FUNCTION_BLOCK E_D_FF_ANY_HYS_TMIN (* Data latch (d) flip flop with a Hysteresis, with a Minimum inter-disposal Time between EO *)
  (* Standard: 61499-1 Annex A; Description: Copyright (c) 2017 fortiss GmbH, HR Agrartechnik GmbH This program and the accompanying materials are made available under the terms of the Eclipse Public License 2.0 which is available at https://www.eclipse.org/legal/epl-2.0/ SPDX-License-Identifier: EPL-2.0 *)
  (* Version 1.0, 2026-05-14, Franz Höpfinger, HR Agrartechnik GmbH, Inital API *)
  PACKAGE logiBUS::signalprocessing::hysteresis;
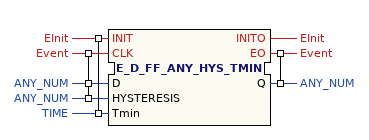
  EVENT_INPUT
    INIT : EInit WITH Tmin; (* Init Request *)
    CLK WITH D, HYSTERESIS; (* Clock *)
  END_EVENT
  EVENT_OUTPUT
    INITO : EInit; (* Init Confirmation *)
    EO WITH Q; (* Triggered if clock results in a change of Q *)
  END_EVENT
  VAR_INPUT
    D : ANY_NUM; (* Value to latch. Must be the same type as Q and HYSTERESIS *)
    HYSTERESIS : ANY_NUM; (* Hysteresis band. Must be the same type as D and Q *)
    Tmin : TIME; (* Minimum inter-arrival time between EI events *)
  END_VAR
  VAR_OUTPUT
    Q : ANY_NUM; (* Latched value. Must be the same type as D and HYSTERESIS *)
  END_VAR
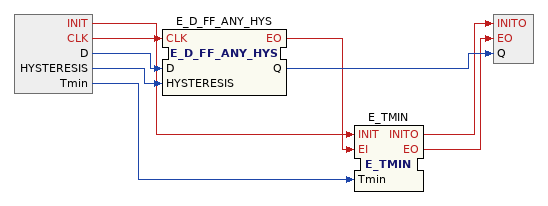
  FBS
    E_D_FF_ANY_HYS : logiBUS::signalprocessing::hysteresis::E_D_FF_ANY_HYS;
    E_TMIN : iec61499::events::E_TMIN;
  END_FBS
  EVENT_CONNECTIONS
    CLK TO E_D_FF_ANY_HYS.CLK;
    INIT TO E_TMIN.INIT;
    E_TMIN.INITO TO INITO;
    E_TMIN.EO TO EO;
    E_D_FF_ANY_HYS.EO TO E_TMIN.EI;
  END_CONNECTIONS
  DATA_CONNECTIONS
    E_D_FF_ANY_HYS.Q TO Q;
    D TO E_D_FF_ANY_HYS.D;
    Tmin TO E_TMIN.Tmin;
    HYSTERESIS TO E_D_FF_ANY_HYS.HYSTERESIS;
  END_CONNECTIONS
END_FUNCTION_BLOCK
